Fanuc KAREL source: kc00047.KL

-- PROVISIONAL review KL for V940-1; original PC SHA256 870bfb7cb577c5f0bf289d3e5c3000bc4667f85546e92ed1ff3fbf0621f81b5c
-- Incomplete behavior may be omitted. Consult companion uncertainty JSON. Do not deploy.
PROGRAM KC00047
%NOLOCKGROUP
BEGIN
  -- V9_ZERO_TABLE_METADATA_HINT layout=0002_ascii; no indexed target words; source/name/runtime held
  -- UNRESOLVED_PC offsets 5-27; opcodes 27,22,22,22,31
  -- UNRESOLVED_PC offsets 32-36; opcodes 7F
END KC00047
